FUNCTION_BLOCK MotorTestSuite EXTENDS TcUnit.FB_TestSuite
VAR_INPUT
END_VAR
VAR_OUTPUT
END_VAR
VAR
END_VAR

METHOD SetEnables
VAR_IN_OUT
    stMotionStage: ST_MotionStage;
END_VAR
stMotionStage.bHardwareEnable := TRUE;
stMotionStage.bLimitBackwardEnable := TRUE;
stMotionStage.bLimitForwardEnable := TRUE;
stMotionStage.bPowerSelf := TRUE;
END_METHOD

METHOD SetGoodState
VAR_IN_OUT
    stPositionState: ST_PositionState;
END_VAR
stPositionState.bMoveOk := TRUE;
stPositionState.bValid := TRUE;
END_METHOD

END_FUNCTION_BLOCK

(* stored: Version 1.1.0.1, ProductVersion 3.1.4022.18
   POU MotorTestSuite: Id {62209a82-679e-47f8-9b5a-ad180dcad4e7}, SpecialFunc None
   Method SetEnables: Id {9a689027-7edb-4bec-9a75-8e1dc053d941}
   Method SetGoodState: Id {b3c6256b-7995-4ca9-aaf3-c136e49e66c8} *)
